(* PLC project Standard IEC Functions, Ambitecs Standard IEC Functions 1.0.0, author Lepekhin Igor *)
(* stored: creationDateTime 2024-09-20T00:00:00, modificationDateTime 2024-11-01T08:00:00 *)

(* Rounding up/down *)
FUNCTION TRUNC : ANY_INT
  VAR_INPUT
    var0 : ANY_REAL;
  END_VAR

END_FUNCTION

(* Conversion to time-of-day *)
FUNCTION DATE_AND_TIME_TO_TIME_OF_DAY : TOD
  VAR_INPUT
    var0 : DT;
  END_VAR

END_FUNCTION

(* Conversion to date *)
FUNCTION DATE_AND_TIME_TO_DATE : DATE
  VAR_INPUT
    var0 : DT;
  END_VAR

END_FUNCTION

(* Absolute number *)
FUNCTION ABS : ANY_NUM
  VAR_INPUT
    var0 : ANY_NUM;
  END_VAR

END_FUNCTION

(* Square root (base 2) *)
FUNCTION SQRT : ANY_REAL
  VAR_INPUT
    var0 : ANY_REAL;
  END_VAR

END_FUNCTION

(* Natural logarithm *)
FUNCTION LN : ANY_REAL
  VAR_INPUT
    var0 : ANY_REAL;
  END_VAR

END_FUNCTION

(* Logarithm to base 10 *)
FUNCTION LOG : ANY_REAL
  VAR_INPUT
    var0 : ANY_REAL;
  END_VAR

END_FUNCTION

(* Exponentiation *)
FUNCTION EXP : ANY_REAL
  VAR_INPUT
    var0 : ANY_REAL;
  END_VAR

END_FUNCTION

(* Sine *)
FUNCTION SIN : ANY_REAL
  VAR_INPUT
    var0 : ANY_REAL;
  END_VAR

END_FUNCTION

(* Cosine *)
FUNCTION COS : ANY_REAL
  VAR_INPUT
    var0 : ANY_REAL;
  END_VAR

END_FUNCTION

(* Tangent *)
FUNCTION TAN : ANY_REAL
  VAR_INPUT
    var0 : ANY_REAL;
  END_VAR

END_FUNCTION

(* Arc sine *)
FUNCTION ASIN : ANY_REAL
  VAR_INPUT
    var0 : ANY_REAL;
  END_VAR

END_FUNCTION

(* Arc cosine *)
FUNCTION ACOS : ANY_REAL
  VAR_INPUT
    var0 : ANY_REAL;
  END_VAR

END_FUNCTION

(* Arc tangent *)
FUNCTION ATAN : ANY_REAL
  VAR_INPUT
    var0 : ANY_REAL;
  END_VAR

END_FUNCTION

(* Addition *)
FUNCTION ADD : ANY_NUM
  VAR_INPUT
    var0 : ANY_NUM;
    var1 : ANY_NUM;
  END_VAR

END_FUNCTION

(* Multiplication *)
FUNCTION MUL : ANY_NUM
  VAR_INPUT
    var0 : ANY_NUM;
    var1 : ANY_NUM;
  END_VAR

END_FUNCTION

(* Subtraction *)
FUNCTION SUB : ANY_NUM
  VAR_INPUT
    var0 : ANY_NUM;
    var1 : ANY_NUM;
  END_VAR

END_FUNCTION

(* Division *)
FUNCTION DIV : ANY_NUM
  VAR_INPUT
    var0 : ANY_NUM;
    var1 : ANY_NUM;
  END_VAR

END_FUNCTION

(* Remainder (modulo) *)
FUNCTION MOD : ANY_INT
  VAR_INPUT
    var0 : ANY_INT;
    var1 : ANY_INT;
  END_VAR

END_FUNCTION

(* Exponent *)
FUNCTION EXPT : ANY_REAL
  VAR_INPUT
    var0 : ANY_REAL;
    var1 : ANY_NUM;
  END_VAR

END_FUNCTION

(* Assignment *)
FUNCTION MOVE : ANY
  VAR_INPUT
    var0 : ANY;
  END_VAR

END_FUNCTION

(* Time addition *)
FUNCTION ADD : TIME
  VAR_INPUT
    var0 : TIME;
    var1 : TIME;
  END_VAR

END_FUNCTION

(* Time addition *)
FUNCTION ADD_TIME : TIME
  VAR_INPUT
    var0 : TIME;
    var1 : TIME;
  END_VAR

END_FUNCTION

(* Time-of-day addition+" "+_("DEPRECATED") *)
FUNCTION ADD : TOD
  VAR_INPUT
    var0 : TOD;
    var1 : TIME;
  END_VAR

END_FUNCTION

(* Time-of-day addition *)
FUNCTION ADD_TOD_TIME : TOD
  VAR_INPUT
    var0 : TOD;
    var1 : TIME;
  END_VAR

END_FUNCTION

(* Date addition+" "+_("DEPRECATED") *)
FUNCTION ADD : DT
  VAR_INPUT
    var0 : DT;
    var1 : TIME;
  END_VAR

END_FUNCTION

(* Date addition *)
FUNCTION ADD_DT_TIME : DT
  VAR_INPUT
    var0 : DT;
    var1 : TIME;
  END_VAR

END_FUNCTION

(* Time multiplication+" "+_("DEPRECATED") *)
FUNCTION MUL : TIME
  VAR_INPUT
    var0 : TIME;
    var1 : ANY_NUM;
  END_VAR

END_FUNCTION

(* Time multiplication *)
FUNCTION MULTIME : TIME
  VAR_INPUT
    var0 : TIME;
    var1 : ANY_NUM;
  END_VAR

END_FUNCTION

(* Time subtraction *)
FUNCTION SUB_TIME : TIME
  VAR_INPUT
    var0 : TIME;
    var1 : TIME;
  END_VAR

END_FUNCTION

(* Time subtraction *)
FUNCTION SUB : TIME
  VAR_INPUT
    var0 : TIME;
    var1 : TIME;
  END_VAR

END_FUNCTION

(* Date subtraction+" "+_("DEPRECATED") *)
FUNCTION SUB : TIME
  VAR_INPUT
    var0 : DATE;
    var1 : DATE;
  END_VAR

END_FUNCTION

(* Date subtraction *)
FUNCTION SUB_DATE_DATE : TIME
  VAR_INPUT
    var0 : DATE;
    var1 : DATE;
  END_VAR

END_FUNCTION

(* Time-of-day subtraction+" "+_("DEPRECATED") *)
FUNCTION SUB : TOD
  VAR_INPUT
    var0 : TOD;
    var1 : TIME;
  END_VAR

END_FUNCTION

(* Time-of-day subtraction *)
FUNCTION SUB_TOD_TIME : TOD
  VAR_INPUT
    var0 : TOD;
    var1 : TIME;
  END_VAR

END_FUNCTION

(* Time-of-day subtraction+" "+_("DEPRECATED") *)
FUNCTION SUB : TIME
  VAR_INPUT
    var0 : TOD;
    var1 : TOD;
  END_VAR

END_FUNCTION

(* Time-of-day subtraction *)
FUNCTION SUB_TOD_TOD : TIME
  VAR_INPUT
    var0 : TOD;
    var1 : TOD;
  END_VAR

END_FUNCTION

(* Date and time subtraction+" "+_("DEPRECATED") *)
FUNCTION SUB : DT
  VAR_INPUT
    var0 : DT;
    var1 : TIME;
  END_VAR

END_FUNCTION

(* Date and time subtraction *)
FUNCTION SUB_DT_TIME : DT
  VAR_INPUT
    var0 : DT;
    var1 : TIME;
  END_VAR

END_FUNCTION

(* Date and time subtraction+" "+_("DEPRECATED") *)
FUNCTION SUB : TIME
  VAR_INPUT
    var0 : DT;
    var1 : DT;
  END_VAR

END_FUNCTION

(* Date and time subtraction *)
FUNCTION SUB_DT_DT : TIME
  VAR_INPUT
    var0 : DT;
    var1 : DT;
  END_VAR

END_FUNCTION

(* Time division+" "+_("DEPRECATED") *)
FUNCTION DIV : TIME
  VAR_INPUT
    var0 : TIME;
    var1 : ANY_NUM;
  END_VAR

END_FUNCTION

(* Time division *)
FUNCTION DIVTIME : TIME
  VAR_INPUT
    var0 : TIME;
    var1 : ANY_NUM;
  END_VAR

END_FUNCTION

(* Shift left *)
FUNCTION SHL : ANY_BIT
  VAR_INPUT
    var0 : ANY_BIT;
    var1 : ANY_INT;  (* Number of bits to be shifted *)
  END_VAR

END_FUNCTION

(* Shift right *)
FUNCTION SHR : ANY_BIT
  VAR_INPUT
    var0 : ANY_BIT;
    var1 : ANY_INT;  (* Number of bits to be shifted *)
  END_VAR

END_FUNCTION

(* Rotate right *)
FUNCTION ROR : ANY_NBIT
  VAR_INPUT
    var0 : ANY_NBIT;
    var1 : ANY_INT;  (* Number of bits to be shifted *)
  END_VAR

END_FUNCTION

(* Rotate left *)
FUNCTION ROL : ANY_NBIT
  VAR_INPUT
    var0 : ANY_NBIT;
    var1 : ANY_INT;  (* Number of bits to be shifted *)
  END_VAR

END_FUNCTION

(* Bitwise AND *)
FUNCTION AND : ANY_BIT
  VAR_INPUT
    var0 : ANY_BIT;
    var1 : ANY_BIT;
  END_VAR

END_FUNCTION

(* Bitwise OR *)
FUNCTION OR : ANY_BIT
  VAR_INPUT
    var0 : ANY_BIT;
    var1 : ANY_BIT;
  END_VAR

END_FUNCTION

(* Bitwise XOR *)
FUNCTION XOR : ANY_BIT
  VAR_INPUT
    var0 : ANY_BIT;
    var1 : ANY_BIT;
  END_VAR

END_FUNCTION

(* Bitwise inverting *)
FUNCTION NOT : ANY_BIT
  VAR_INPUT
    var0 : ANY_BIT;
  END_VAR

END_FUNCTION

(* Binary selection (1 of 2) *)
FUNCTION SEL : ANY
  VAR_INPUT
    var0 : BOOL;  (* Selection out of 2 inputs (gate) *)
    var1 : ANY;
    var2 : ANY;
  END_VAR

END_FUNCTION

(* Maximum *)
FUNCTION MAX : ANY
  VAR_INPUT
    var0 : ANY;
    var1 : ANY;
  END_VAR

END_FUNCTION

(* Minimum *)
FUNCTION MIN : ANY
  VAR_INPUT
    var0 : ANY;
    var1 : ANY;
  END_VAR

END_FUNCTION

(* Limitation *)
FUNCTION LIMIT : ANY
  VAR_INPUT
    var0 : ANY;  (* Minimum value for limitation *)
    var1 : ANY;
    var2 : ANY;  (* Maximum value for limitation *)
  END_VAR

END_FUNCTION

(* Multiplexer (select 1 of N) *)
FUNCTION MUX : ANY
  VAR_INPUT
    var0 : ANY_INT;  (* Selection out of n inputs *)
    var1 : ANY;
    var2 : ANY;
  END_VAR

END_FUNCTION

(* Greater than *)
FUNCTION GT : BOOL
  VAR_INPUT
    var0 : ANY;
    var1 : ANY;
  END_VAR

END_FUNCTION

(* Greater than or equal to *)
FUNCTION GE : BOOL
  VAR_INPUT
    var0 : ANY;
    var1 : ANY;
  END_VAR

END_FUNCTION

(* Equal to *)
FUNCTION EQ : BOOL
  VAR_INPUT
    var0 : ANY;
    var1 : ANY;
  END_VAR

END_FUNCTION

(* Less than *)
FUNCTION LT : BOOL
  VAR_INPUT
    var0 : ANY;
    var1 : ANY;
  END_VAR

END_FUNCTION

(* Less than or equal to *)
FUNCTION LE : BOOL
  VAR_INPUT
    var0 : ANY;
    var1 : ANY;
  END_VAR

END_FUNCTION

(* Not equal to *)
FUNCTION NE : BOOL
  VAR_INPUT
    var0 : ANY;
    var1 : ANY;
  END_VAR

END_FUNCTION

(* Length of string *)
FUNCTION LEN : INT
  VAR_INPUT
    var0 : STRING;
  END_VAR

END_FUNCTION

(* string left of *)
FUNCTION LEFT : STRING
  VAR_INPUT
    var0 : STRING;
    var1 : ANY_INT;  (* Left position within character string *)
  END_VAR

END_FUNCTION

(* string right of *)
FUNCTION RIGHT : STRING
  VAR_INPUT
    var0 : STRING;
    var1 : ANY_INT;  (* Left position within character string *)
  END_VAR

END_FUNCTION

(* string from the middle *)
FUNCTION MID : STRING
  VAR_INPUT
    var0 : STRING;
    var1 : ANY_INT;  (* Left position within character string *)
    var2 : ANY_INT;  (* Position within character string *)
  END_VAR

END_FUNCTION

(* Concatenation *)
FUNCTION CONCAT : STRING
  VAR_INPUT
    var0 : STRING;
    var1 : STRING;
  END_VAR

END_FUNCTION

(* Time concatenation *)
FUNCTION CONCAT_DATE_TOD : DT
  VAR_INPUT
    var0 : DATE;
    var1 : TOD;
  END_VAR

END_FUNCTION

(* Insertion (into) *)
FUNCTION INSERT : STRING
  VAR_INPUT
    var0 : STRING;
    var1 : STRING;
    var2 : ANY_INT;  (* Position within character string *)
  END_VAR

END_FUNCTION

(* Deletion (within) *)
FUNCTION DELETE : STRING
  VAR_INPUT
    var0 : STRING;
    var1 : ANY_INT;  (* Left position within character string *)
    var2 : ANY_INT;  (* Position within character string *)
  END_VAR

END_FUNCTION

(* Replacement (within) *)
FUNCTION REPLACE : STRING
  VAR_INPUT
    var0 : STRING;
    var1 : STRING;
    var2 : ANY_INT;  (* Left position within character string *)
    var3 : ANY_INT;  (* Position within character string *)
  END_VAR

END_FUNCTION

(* Find position *)
FUNCTION FIND : INT
  VAR_INPUT
    var0 : STRING;
    var1 : STRING;
  END_VAR

END_FUNCTION
